FUNCTION_BLOCK p_InitVar
VAR_INPUT
END_VAR
VAR_OUTPUT
END_VAR
VAR
	tEnvStabSort: INT;
END_VAR

fbAct1.stParam.xPresenceSensIn:=TRUE;
fbAct1.stParam.xPresenceSensOut:=TRUE;
fbAct1.stParam.tTimeOut:=T#10S;
fbAct1.stParam.tMoveInTimeDelay:=T#1.5S;
fbAct1.stParam.tMoveOutTimeDelay:=T#1.5S;

fbAct2.stParam.xPresenceSensIn:=TRUE;
fbAct2.stParam.xPresenceSensOut:=TRUE;
fbAct2.stParam.tTimeOut:=T#10S;
fbAct2.stParam.tMoveInTimeDelay:=T#1.5S;
fbAct2.stParam.tMoveOutTimeDelay:=T#1.5S;

fbAct3.stParam.xPresenceSensIn:=FALSE;
fbAct3.stParam.xPresenceSensOut:=TRUE;
fbAct3.stParam.tTimeOut:=T#10S;
fbAct3.stParam.tMoveInTimeDelay:=T#3S;
fbAct3.stParam.tMoveOutTimeDelay:=T#1.5S;

stParam.stStatus.eMMA:=Init;

END_FUNCTION_BLOCK

(* stored: Version 1.1.0.1, ProductVersion 3.1.4020.6
   POU p_InitVar: Id {202cf7ca-6c5b-44f0-9a22-b821172721e6}, SpecialFunc None *)
